FUNCTION_BLOCK Resource3
  (* Version 1.0, 2008-11-12, Goran Cengic, Chalmers *)
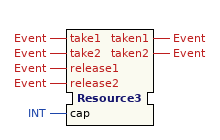
  EVENT_INPUT
    take1;
    take2;
    release1;
    release2;
  END_EVENT
  EVENT_OUTPUT
    taken1;
    taken2;
  END_EVENT
  VAR_INPUT
    cap : INT;
  END_VAR
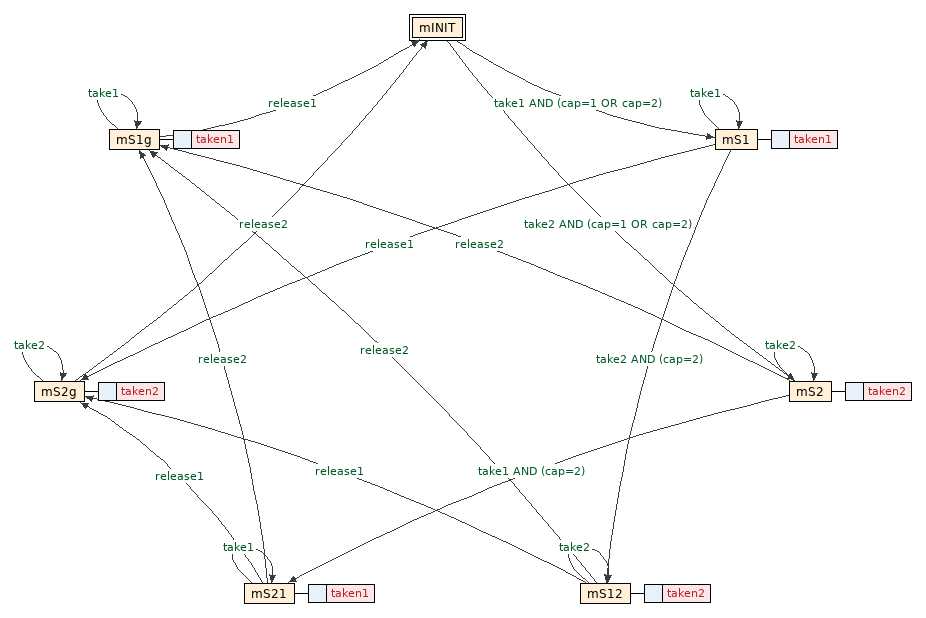
  EC_STATES
    mINIT;
    mS1 : -> taken1;
    mS2 : -> taken2;
    mS12 : -> taken2;
    mS21 : -> taken1;
    mS2g : -> taken2;
    mS1g : -> taken1;
  END_STATES
  EC_TRANSITIONS
    mINIT TO mS1 := take1 AND (cap=1 OR cap=2);
    mS1 TO mS1 := take1;
    mS1 TO mS2g := release1;
    mS2g TO mS2g := take2;
    mS2g TO mINIT := release2;
    mINIT TO mS2 := take2 AND (cap=1 OR cap=2);
    mS2 TO mS2 := take2;
    mS2 TO mS1g := release2;
    mS1g TO mS1g := take1;
    mS1g TO mINIT := release1;
    mS1 TO mS12 := take2 AND (cap=2);
    mS12 TO mS12 := take2;
    mS12 TO mS2g := release1;
    mS12 TO mS1g := release2;
    mS2 TO mS21 := take1 AND (cap=2);
    mS21 TO mS21 := take1;
    mS21 TO mS1g := release2;
    mS21 TO mS2g := release1;
  END_TRANSITIONS
END_FUNCTION_BLOCK
